{attribute 'GeneratedUsingTerminal: EK1100-0000-0018'}
{attribute addProperty BoxType "EK1100-0000-0018"}
{attribute addProperty Id "Beckhoff_APS4xxxEK1122Beckhoff_APS4xxxEK1122_73545D62284A_0002_APS4322_5000_0017APS4322_748FE0C1320"}
{attribute addProperty CRC "686462767"}
{attribute addProperty Size "604"}
TYPE Beckhoff_APS4xxx_28EA972F EXTENDS EK1100_AB5A9467 :
STRUCT
	{attribute addProperty Name "Beckhoff_APS4xxxEK1122"}
	Beckhoff_APS4xxxEK1122 : Beckhoff_APS4xxxEK1122_73545D62;
	{attribute addProperty Name "A_0002_APS4322_5000_0017"}
	A_0002_APS4322_5000_0017 : APS4322_748FE0C1;
END_STRUCT
END_TYPE

(* stored: Version 1.2.0.0, ProductVersion 3.1.4024.9
   DUT Beckhoff_APS4xxx_28EA972F: Id {f6899d7d-1af9-4201-98a2-011ad7f117fa} *)
